// TIA Portal V15.1 export
// export: Created 2024-06-21T08:41:08.8202615Z, ExportSetting WithDefaults, DisplayName Totally Integrated Automation Portal, DisplayVersion V15.1 Update 5, DisplayName TIA Portal Openness, DisplayVersion V15.1 Update 5, DisplayName SINAMICS Startdrive Advanced, DisplayVersion V15.1, DisplayName G130, G150, S120, S150, SINAMICS MV, S210, DisplayVersion V15.1, DisplayName G110M, G120, G120C, G120D, G120P, DisplayVersion V15.1, DisplayName STEP 7 Professional, DisplayVersion V15.1 Update 5, DisplayName STEP 7 Safety, DisplayVersion V15.1, DisplayName WinCC Professional, DisplayVersion V15.1 Update 5, DisplayName SIMATIC Visualization Architect, DisplayVersion V15.1
FUNCTION "LGBProdStartStop-Config" : Void   // FC6645, FBD
TITLE = LGBProdStartStop-Config
{ S7_Optimized_Access := 'FALSE' }
AUTHOR : VCC
FAMILY : Control
NAME : Bit2Word
VERSION : 1.0
// stored: AutoNumber false, IsIECCheckEnabled false, SetENOAutomatically False, UDAEnableTagReadback false
   VAR_INPUT
      C_AndonHCallDirectStop : Bool;   // By Andon Human Call direct stop of the productionline
      C_AndonECallDirectStop : Bool;   // By Andon Equipment Call direct stop of the productionline
      C_AndonMCallDirectStop : Bool;   // By Andon Material Call direct stop of the productionline
      C_DefaultGapsIsAllowed : Bool;   // Default GAPS allowed is active
   END_VAR
   VAR_IN_OUT
      IO_Config : "ProdStartStopConfig";   // Config
   END_VAR
BEGIN

REGION Network 1: **** 1 Inputs **** Config
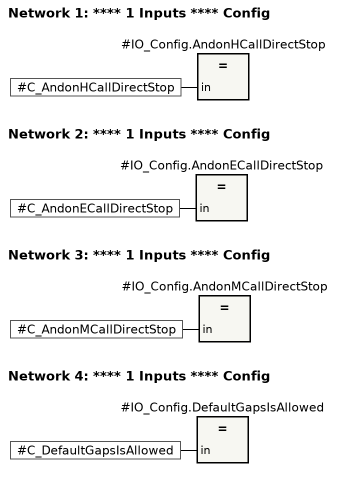
   #IO_Config.AndonHCallDirectStop := #C_AndonHCallDirectStop;
END_REGION

REGION Network 2: **** 1 Inputs **** Config
   #IO_Config.AndonECallDirectStop := #C_AndonECallDirectStop;
END_REGION

REGION Network 3: **** 1 Inputs **** Config
   #IO_Config.AndonMCallDirectStop := #C_AndonMCallDirectStop;
END_REGION

REGION Network 4: **** 1 Inputs **** Config
   #IO_Config.DefaultGapsIsAllowed := #C_DefaultGapsIsAllowed;
END_REGION
END_FUNCTION
